SUBAPPLICATION Gripper (* Subapplication Type *)
  (* Standard: 61499-2 *)
  (* Version 1.0, 2018-07-10, az *)
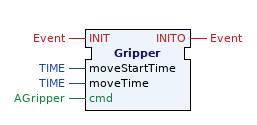
  EVENT_INPUT
    INIT;
  END_EVENT
  EVENT_OUTPUT
    INITO;
  END_EVENT
  VAR_INPUT
    moveStartTime : TIME;
    moveTime : TIME;
  END_VAR
  SOCKETS
    cmd : AGripper;
  END_SOCKETS
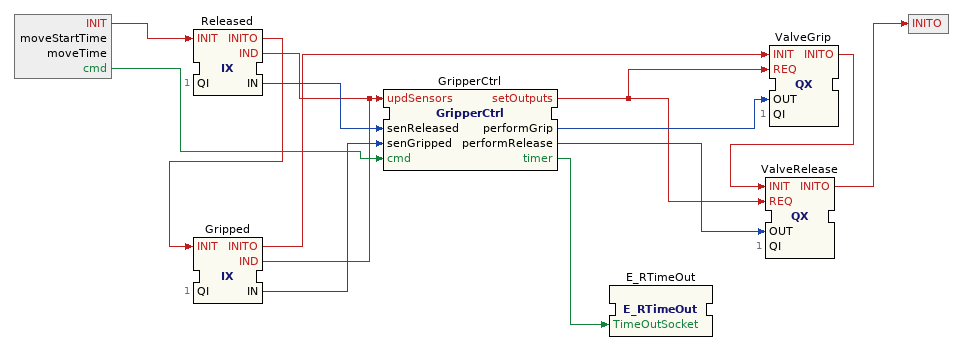
  FBS
    ValveRelease : QX(QI := 1);
    Released : IX(QI := 1);
    Gripped : IX(QI := 1);
    ValveGrip : QX(QI := 1);
    E_RTimeOut : E_RTimeOut;
    GripperCtrl : GripperCtrl;
  END_FBS
  EVENT_CONNECTIONS
    ValveGrip.INITO TO ValveRelease.INIT;
    Released.INITO TO Gripped.INIT;
    Gripped.INITO TO ValveGrip.INIT;
    INIT TO Released.INIT;
    ValveRelease.INITO TO INITO;
    Released.IND TO GripperCtrl.updSensors;
    Gripped.IND TO GripperCtrl.updSensors;
    GripperCtrl.setOutputs TO ValveRelease.REQ;
    GripperCtrl.setOutputs TO ValveGrip.REQ;
  END_CONNECTIONS
  DATA_CONNECTIONS
    Released.IN TO GripperCtrl.senReleased;
    Gripped.IN TO GripperCtrl.senGripped;
    GripperCtrl.performGrip TO ValveGrip.OUT;
    GripperCtrl.performRelease TO ValveRelease.OUT;
  END_CONNECTIONS
  ADAPTER_CONNECTIONS
    GripperCtrl.timer TO E_RTimeOut.TimeOutSocket;
    cmd TO GripperCtrl.cmd;
  END_CONNECTIONS
END_SUBAPPLICATION
